
// ===== library: MasterCopy "FB_REOComm" =====

// folder: 04_Heating

FUNCTION_BLOCK "FB_REOComm"   // FB53, SCL
{ S7_Optimized_Access := 'TRUE' }
VERSION : 0.1
   VAR_INPUT
      i_wParameterAdr : Word;   // Address of the parameter to read or write in HEX
      i_wNewValue : Word;   // Value to write to the parameter
      i_wSendStrom : Word;   // Current setpoint (to be sent to REO) 16-Bit 100 % = FFFF H
      i_wSendSpannung : Word;   // Voltage setpoint (to be sent to REO) 16-Bit 100 % = FFFF H
      i_wSendLeistung : Word;   // Power setpoint (to be sent to REO) 16-Bit 100 % = FFFF H
      i_xCurrentPowerMode : Bool;   // 0 = current mode, 1 = power mode
      i_xSendParameter : Bool;   // Trigger to start send parameter sequence
      i_xReadParameter : Bool;   // Trigger to start read parameter sequence
      i_xFreigabeHeiz : Bool;   // Heating enable signal
      i_xResetREO : Bool;   // Trigger to reset REO via parameter mode
      i_xConfigMDW700 : Bool;   // Configuration bit to use the the rigth status byte structure
      i_xConfigWRB : Bool;   // Configuration bit to use the the rigth status byte structure
   END_VAR
   VAR_OUTPUT
      o_REOStatus : "typeREOStatus";   // Structure with REO state and error info
      o_awHWRead : Array[1..4] of Word;   // Read buffer from REO (from DPRD_DAT) [4 WORDs]
      o_wStatusSend : Word;   // Status from the DPWR_DAT call (communication status)
      o_wStatusRead : Word;   // Status from the DPRD_DAT call (communication status)
      o_wReadStrom : Word;   // Measured current from REO (Word 3) Istwert Strom 16 Bit 100% = 8000 H
      o_wReadSpannung : Word;   // Measured voltage from REO (Word 2) Istwert Spannung 16 Bit 100% = 8000 H
      o_wReadLeistung : Word;   // Measured power from REO (Word 2) Istwert Leistung 16 Bit 100% = 4000H
      o_wReadedParameter : Word;   // The parameter value read from REO
      o_xNormalbetrieb : Bool;   // Output for normal operation status
      o_xParameterbetrieb : Bool;   // Output for parameter operation status
      o_xBusy : Bool;   // TRUE when operation in progress
      o_xReadDone : Bool;   // TRUE when Read parameter sequence is done
      o_xResetDone : Bool;   // TRUE when Reset completed successfully
      o_xSendDone : Bool;   // TRUE when Send parameter sequence is done
      o_xError : Bool;   // TRUE if timeout or failure occurred
   END_VAR
   VAR
      TON_TimeResponseOut : TON_TIME;   // Timeout watchdog (e.g., to prevent stuck communication)
      stat_awHWSend : Array[1..4] of Word;   // Internal buffer for writing to REO [4 WORDs]
      iStateWriteParameter : Int;   // Internal state for the write paramter state machine
      iStateReadParameter : Int;   // Internal state for the read paramter state machine
      iStateResetREO : Int;   // Internal state for the reset state machine
      xNormalbetrieb : Bool := TRUE;   // Normal operation mode (standard REO heating control)
      xParameterbetrieb : Bool;   // Parameter operation mode (for parameter read/write/reset)
   END_VAR
   VAR_TEMP
      temp_bySteuerWortError : Byte;
   END_VAR
   VAR CONSTANT
      cCODE : Word := 16#C0DE;   // Constant C0DEH, used in REO protocol as signature
   END_VAR
BEGIN
   (********************************************************************************************************
   Author:     IK
   Date:       2025-04
   Version:    1.1
   *********************************************************************************************************
   Purpose:
   Implements normal mode and parameter mode communication with REO devices via Profinet
   It uses Siemens functions DPRD_DAT and DPWR_DAT to read and write registers from REO
   It also writes status / diagnostic information from REO
   When sending, it sends a sequence of commands: Write Enable, Parameter Write, Release Write Enable,
   Read value and waits for confirmation from the device.
   Use REO Profinet description information documentation to get parameter addresses in Hex

   *********************************************************************************************************
   Modification notes:
   Date:              Name:            Description
   2025-05-19         IK               Added 2 vars: i_xConfigMDW700, i_xConfigWRB
                                       Updated "REO status byte read" block
   *)
   // === Switch to parameter mode when trigger is active ===
   IF (#i_xResetREO
     OR #i_xReadParameter
     OR #i_xSendParameter)
     AND #xNormalbetrieb
   THEN
     // Switch from normal to parameter mode
     #xNormalbetrieb := FALSE;
     #xParameterbetrieb := TRUE;
     #o_xReadDone := FALSE;
     #o_xSendDone := FALSE;
     #o_xResetDone := FALSE;
     #o_xError := FALSE;
   END_IF;

   // === Timeout monitoring for REO system response (5 seconds) ===
   #TON_TimeResponseOut(IN := #xParameterbetrieb
                        AND (#iStateReadParameter <> 0
                        OR #iStateWriteParameter <> 0
                        OR #iStateResetREO <> 0),
                        PT := T#5s);

   IF #TON_TimeResponseOut.Q THEN
     // Timeout: cancel communication and return to normal mode
     #iStateReadParameter := 0;
     #xParameterbetrieb := FALSE;
     #xNormalbetrieb := TRUE;
     #o_xBusy := FALSE;
     #o_xReadDone := FALSE;
     #o_xSendDone := FALSE;
     #o_xError := TRUE;
   END_IF;

   IF #xNormalbetrieb THEN
     //Read from REO
     #o_wStatusRead := INT_TO_WORD(DPRD_DAT(LADDR := "REO_Thyristorsteller_(Phasenanschnitt)~IN_OUT:____8_bytes_1", RECORD => #o_awHWRead));

     IF #i_xCurrentPowerMode THEN
       // Read power and current
       #o_wReadLeistung := #o_awHWRead[2]; // actual power: 4000 = 16384 = 100% max REO power
       #o_wReadStrom := #o_awHWRead[3];    // actual current: 8000 = 32768 = 100% max REO current
     ELSE
       // Read voltage and current
       #o_wReadSpannung := #o_awHWRead[2]; // actual voltage: 8000 = 32768 = 100% max REO voltage
       #o_wReadStrom := #o_awHWRead[3];    // actual current: 8000 = 32768 = 100% max REO current
     END_IF;


     // REO status byte read - read and interpret status byte
     // (various REO operating or fault states depending on error code)
     #temp_bySteuerWortError := #o_awHWRead[4].%B1;
     IF #i_xConfigMDW700 THEN
       CASE #temp_bySteuerWortError OF
         16#00:  // Device not responding
           #o_REOStatus.xReagiertNicht := TRUE;
           #o_REOStatus.xBetriebsbereit := FALSE;
           #o_REOStatus.xParametermodus := FALSE;
           #o_REOStatus.xÜbertemperatur := FALSE;
           #o_REOStatus.xÜberstrom := FALSE;
           #o_REOStatus.xÜberspannung := FALSE;
           #o_REOStatus.xSpitzenStrom := FALSE;
           #o_REOStatus.xUnknowCode := FALSE;
           #o_REOStatus.byREOFehlerCode := #temp_bySteuerWortError;
         16#A5:  // Device ready for operation
           #o_REOStatus.xReagiertNicht := FALSE;
           #o_REOStatus.xBetriebsbereit := TRUE;
           #o_REOStatus.xParametermodus := FALSE;
           #o_REOStatus.xÜbertemperatur := FALSE;
           #o_REOStatus.xÜberstrom := FALSE;
           #o_REOStatus.xÜberspannung := FALSE;
           #o_REOStatus.xSpitzenStrom := FALSE;
           #o_REOStatus.xUnknowCode := FALSE;
           #o_REOStatus.byREOFehlerCode := #temp_bySteuerWortError;
         16#C0:  // Feedback: parameter mode
           #o_REOStatus.xReagiertNicht := FALSE;
           #o_REOStatus.xBetriebsbereit := FALSE;
           #o_REOStatus.xParametermodus := TRUE;
           #o_REOStatus.xÜbertemperatur := FALSE;
           #o_REOStatus.xÜberstrom := FALSE;
           #o_REOStatus.xÜberspannung := FALSE;
           #o_REOStatus.xSpitzenStrom := FALSE;
           #o_REOStatus.xUnknowCode := FALSE;
           #o_REOStatus.byREOFehlerCode := #temp_bySteuerWortError;
         16#70:  // ERROR HOT, overtemperature
           #o_REOStatus.xReagiertNicht := FALSE;
           #o_REOStatus.xBetriebsbereit := FALSE;
           #o_REOStatus.xParametermodus := FALSE;
           #o_REOStatus.xÜbertemperatur := TRUE;
           #o_REOStatus.xÜberstrom := FALSE;
           #o_REOStatus.xÜberspannung := FALSE;
           #o_REOStatus.xSpitzenStrom := FALSE;
           #o_REOStatus.xUnknowCode := FALSE;
           #o_REOStatus.byREOFehlerCode := #temp_bySteuerWortError;
         16#58:  // ERROR OL, overcurrent
           #o_REOStatus.xReagiertNicht := FALSE;
           #o_REOStatus.xBetriebsbereit := FALSE;
           #o_REOStatus.xParametermodus := FALSE;
           #o_REOStatus.xÜbertemperatur := FALSE;
           #o_REOStatus.xÜberstrom := TRUE;
           #o_REOStatus.xÜberspannung := FALSE;
           #o_REOStatus.xSpitzenStrom := FALSE;
           #o_REOStatus.xUnknowCode := FALSE;
           #o_REOStatus.byREOFehlerCode := #temp_bySteuerWortError;
         16#05:  // ERROR UL, overvoltage
           #o_REOStatus.xReagiertNicht := FALSE;
           #o_REOStatus.xBetriebsbereit := FALSE;
           #o_REOStatus.xParametermodus := FALSE;
           #o_REOStatus.xÜbertemperatur := FALSE;
           #o_REOStatus.xÜberstrom := FALSE;
           #o_REOStatus.xÜberspannung := TRUE;
           #o_REOStatus.xSpitzenStrom := FALSE;
           #o_REOStatus.xUnknowCode := FALSE;
           #o_REOStatus.byREOFehlerCode := #temp_bySteuerWortError;
         ELSE  // Unknown status code
           #o_REOStatus.xReagiertNicht := FALSE;
           #o_REOStatus.xBetriebsbereit := FALSE;
           #o_REOStatus.xParametermodus := FALSE;
           #o_REOStatus.xÜbertemperatur := FALSE;
           #o_REOStatus.xÜberstrom := FALSE;
           #o_REOStatus.xÜberspannung := FALSE;
           #o_REOStatus.xSpitzenStrom := FALSE;
           #o_REOStatus.xUnknowCode := TRUE;
           #o_REOStatus.byREOFehlerCode := #temp_bySteuerWortError;
       END_CASE;
     ELSIF #i_xConfigWRB THEN
       CASE #temp_bySteuerWortError OF
         16#00:  // Device not responding
           #o_REOStatus.xReagiertNicht := TRUE;
           #o_REOStatus.xBetriebsbereit := FALSE;
           #o_REOStatus.xParametermodus := FALSE;
           #o_REOStatus.xÜbertemperatur := FALSE;
           #o_REOStatus.xÜberstrom := FALSE;
           #o_REOStatus.xÜberspannung := FALSE;
           #o_REOStatus.xSpitzenStrom := FALSE;
           #o_REOStatus.xUnknowCode := FALSE;
           #o_REOStatus.byREOFehlerCode := #temp_bySteuerWortError;
         16#A5:  // Device ready for operation
           #o_REOStatus.xReagiertNicht := FALSE;
           #o_REOStatus.xBetriebsbereit := TRUE;
           #o_REOStatus.xParametermodus := FALSE;
           #o_REOStatus.xÜbertemperatur := FALSE;
           #o_REOStatus.xÜberstrom := FALSE;
           #o_REOStatus.xÜberspannung := FALSE;
           #o_REOStatus.xSpitzenStrom := FALSE;
           #o_REOStatus.xUnknowCode := FALSE;
           #o_REOStatus.byREOFehlerCode := #temp_bySteuerWortError;
         16#C0:  // Feedback: parameter mode
           #o_REOStatus.xReagiertNicht := FALSE;
           #o_REOStatus.xBetriebsbereit := FALSE;
           #o_REOStatus.xParametermodus := TRUE;
           #o_REOStatus.xÜbertemperatur := FALSE;
           #o_REOStatus.xÜberstrom := FALSE;
           #o_REOStatus.xÜberspannung := FALSE;
           #o_REOStatus.xSpitzenStrom := FALSE;
           #o_REOStatus.xUnknowCode := FALSE;
           #o_REOStatus.byREOFehlerCode := #temp_bySteuerWortError;
         16#70:  // ERROR HOT, overtemperature
           #o_REOStatus.xReagiertNicht := FALSE;
           #o_REOStatus.xBetriebsbereit := FALSE;
           #o_REOStatus.xParametermodus := FALSE;
           #o_REOStatus.xÜbertemperatur := TRUE;
           #o_REOStatus.xÜberstrom := FALSE;
           #o_REOStatus.xÜberspannung := FALSE;
           #o_REOStatus.xSpitzenStrom := FALSE;
           #o_REOStatus.xUnknowCode := FALSE;
           #o_REOStatus.byREOFehlerCode := #temp_bySteuerWortError;
         16#58:  // ERROR OL, overcurrent
           #o_REOStatus.xReagiertNicht := FALSE;
           #o_REOStatus.xBetriebsbereit := FALSE;
           #o_REOStatus.xParametermodus := FALSE;
           #o_REOStatus.xÜbertemperatur := FALSE;
           #o_REOStatus.xÜberstrom := TRUE;
           #o_REOStatus.xÜberspannung := FALSE;
           #o_REOStatus.xSpitzenStrom := FALSE;
           #o_REOStatus.xUnknowCode := FALSE;
           #o_REOStatus.byREOFehlerCode := #temp_bySteuerWortError;
         16#37:  // ERROR UL, overvoltage
           #o_REOStatus.xReagiertNicht := FALSE;
           #o_REOStatus.xBetriebsbereit := FALSE;
           #o_REOStatus.xParametermodus := FALSE;
           #o_REOStatus.xÜbertemperatur := FALSE;
           #o_REOStatus.xÜberstrom := FALSE;
           #o_REOStatus.xÜberspannung := TRUE;
           #o_REOStatus.xSpitzenStrom := FALSE;
           #o_REOStatus.xUnknowCode := FALSE;
           #o_REOStatus.byREOFehlerCode := #temp_bySteuerWortError;
         16#57:  // ERROR PEAK, peak current
           #o_REOStatus.xReagiertNicht := FALSE;
           #o_REOStatus.xBetriebsbereit := FALSE;
           #o_REOStatus.xParametermodus := FALSE;
           #o_REOStatus.xÜbertemperatur := FALSE;
           #o_REOStatus.xÜberstrom := FALSE;
           #o_REOStatus.xÜberspannung := TRUE;
           #o_REOStatus.xSpitzenStrom := TRUE;
           #o_REOStatus.xUnknowCode := FALSE;
           #o_REOStatus.byREOFehlerCode := #temp_bySteuerWortError;
         ELSE  // Unknown status code
           #o_REOStatus.xReagiertNicht := FALSE;
           #o_REOStatus.xBetriebsbereit := FALSE;
           #o_REOStatus.xParametermodus := FALSE;
           #o_REOStatus.xÜbertemperatur := FALSE;
           #o_REOStatus.xÜberstrom := FALSE;
           #o_REOStatus.xÜberspannung := FALSE;
           #o_REOStatus.xSpitzenStrom := FALSE;
           #o_REOStatus.xUnknowCode := TRUE;
           #o_REOStatus.byREOFehlerCode := #temp_bySteuerWortError;
       END_CASE;
     ELSE
       ;   // Optional default: do nothing
     END_IF;

     IF #i_xCurrentPowerMode THEN // Set setpoints and send to REO
       // Power / current mode
       IF #i_xFreigabeHeiz THEN
         // Send voltage and current setpoint, activate Bit 2 (enable)
         #stat_awHWSend[1] := 16#0000;           // must be 0000
         #stat_awHWSend[2] := #i_wSendLeistung;  // setpoint power: 16#FFFF = 65535 = 100% max REO power
         #stat_awHWSend[3] := #i_wSendStrom;     // setpoint current: 16#FFFF = 65535 = 100% REO current
         #stat_awHWSend[4] := 16#4004;           // enable on Bit 2
       ELSE
         // Set everything to 0, disable heating
         #stat_awHWSend[1] := 16#0000;
         #stat_awHWSend[2] := 16#0000;
         #stat_awHWSend[3] := 16#0000;
         #stat_awHWSend[4] := 16#0000;
       END_IF;
     ELSE
       // Voltage / current mode
       IF #i_xFreigabeHeiz THEN
         // Send voltage and current setpoint, activate Bit 2 (enable)
         #stat_awHWSend[1] := 16#0000;           // must be 0000
         #stat_awHWSend[2] := #i_wSendSpannung;  // setpoint voltage: 16#FFFF = 65535 = 100% REO voltage
         #stat_awHWSend[3] := #i_wSendStrom;     // setpoint current: 16#FFFF = 65535 = 100% REO current
         #stat_awHWSend[4] := 16#4004;           // enable on Bit 2
       ELSE
         // Set everything to 0, disable heating
         #stat_awHWSend[1] := 16#0000;
         #stat_awHWSend[2] := 16#0000;
         #stat_awHWSend[3] := 16#0000;
         #stat_awHWSend[4] := 16#0000;           // disable
       END_IF;
     END_IF;


     // Send to REO over DPWR_DAT
     #o_wStatusSend := INT_TO_WORD(DPWR_DAT(LADDR := "REO_Thyristorsteller_(Phasenanschnitt)~IN_OUT:____8_bytes_1", RECORD := #stat_awHWSend));

   ELSIF #xParameterbetrieb THEN
     #o_wStatusRead := INT_TO_WORD(DPRD_DAT(LADDR := "REO_Thyristorsteller_(Phasenanschnitt)~IN_OUT:____8_bytes_1", RECORD => #o_awHWRead));
     CASE #iStateResetREO OF
       0: //Idle: wait for trigger
         IF #i_xResetREO THEN
           // Enable write permission
           #stat_awHWSend[1] := 16#0000;
           #stat_awHWSend[2] := #cCODE;    // Address write key = C0DEH
           #stat_awHWSend[3] := 16#B5C9;   // Write-key for enable = B5E7H
           #stat_awHWSend[4] := 16#8000;   // Mode bits: set mode bit = 1
           #o_wStatusSend := INT_TO_WORD(DPWR_DAT(LADDR := "REO_Thyristorsteller_(Phasenanschnitt)~IN_OUT:____8_bytes_1", RECORD := #stat_awHWSend));
           #iStateResetREO := 1;
           #o_xBusy := TRUE;
         END_IF;

       1: // Wait for confirmation and write reset parameter
         IF #o_awHWRead[1] = 16#0000
           AND #o_awHWRead[2] = #cCODE
           AND #o_awHWRead[3] = 16#B5C9
           AND #o_awHWRead[4] = #cCODE
         THEN
           #stat_awHWSend[1] := 16#0000;
           #stat_awHWSend[2] := 16#9400;   // Address write key = C0DEH
           #stat_awHWSend[3] := 16#C009;   // Write-key for enable = B5E7H
           #stat_awHWSend[4] := 16#8000;   // Mode bits: set mode bit = 1
           #o_wStatusSend := INT_TO_WORD(DPWR_DAT(LADDR := "REO_Thyristorsteller_(Phasenanschnitt)~IN_OUT:____8_bytes_1", RECORD := #stat_awHWSend));
           #iStateResetREO := 2;
         END_IF;

       2: // Wait for confirmation and stop parameter mode
         IF #o_awHWRead[1] = 16#0000
           AND #o_awHWRead[2] = 16#0000
           AND #o_awHWRead[3] = 16#0000
           AND #o_awHWRead[4] = #cCODE
         THEN
           #iStateResetREO := 0;
           #xParameterbetrieb := FALSE;
           #xNormalbetrieb := TRUE;
           #o_xBusy := FALSE;
           #o_xResetDone := TRUE;
         END_IF;
     END_CASE;

     // State machine: read parameter only
     CASE #iStateReadParameter OF
       0: // Idle: wait for trigger and read the parameter
         IF #i_xReadParameter THEN
           #stat_awHWSend[1] := 16#0000;
           #stat_awHWSend[2] := #i_wParameterAdr;
           #stat_awHWSend[3] := 16#0000;
           #stat_awHWSend[4] := 16#8000;
           #o_wStatusSend := INT_TO_WORD(DPWR_DAT(LADDR := "REO_Thyristorsteller_(Phasenanschnitt)~IN_OUT:____8_bytes_1", RECORD := #stat_awHWSend));
           #iStateReadParameter := 1;
           #o_xBusy := TRUE;
         END_IF;

       1: //Wait for response and get the parameter
         IF #o_awHWRead[1] = 16#0000
           AND #o_awHWRead[2] = #i_wParameterAdr
           AND #o_awHWRead[4] = #cCODE
         THEN
           #o_wReadedParameter := #o_awHWRead[3];
           #iStateReadParameter := 0;
           #xParameterbetrieb := FALSE;
           #xNormalbetrieb := TRUE;
           #o_xBusy := FALSE;
           #o_xReadDone := TRUE;
         END_IF;
     END_CASE;

     // State machine: write parameter
     CASE #iStateWriteParameter OF
       0:  // Idle: wait for trigger
         IF #i_xSendParameter THEN
           // Step 1: Send Schreibfreigabe (Write Enable)
           #stat_awHWSend[1] := 16#0000;
           #stat_awHWSend[2] := #cCODE;   // Adresse Schreibschlüssel = C0DEH
           #stat_awHWSend[3] := 16#B5E7;   // Write-key for enable = B5E7H
           #stat_awHWSend[4] := 16#8000;   // Mode bits: set mode bit = 1
           #o_wStatusSend := INT_TO_WORD(DPWR_DAT(LADDR := "REO_Thyristorsteller_(Phasenanschnitt)~IN_OUT:____8_bytes_1", RECORD := #stat_awHWSend));
           #iStateWriteParameter := 1;
           #o_xBusy := TRUE;
         END_IF;

       1:  // Waiting for confirmation of Schreibfreigabe and then send parameter
         IF #o_awHWRead[1] = 16#0000
           AND #o_awHWRead[2] = #cCODE
           AND #o_awHWRead[3] = 16#B5E7
           AND #o_awHWRead[4] = #cCODE
         THEN
           #stat_awHWSend[1] := 16#0000;
           #stat_awHWSend[2] := #i_wParameterAdr OR 16#8000; // Word 2: parameter address with R/W bit; set R/W = 1 (write), for example:
           #stat_awHWSend[3] := #i_wNewValue;  // The new parameter value
           #stat_awHWSend[4] := 16#8000;      // Mode bits (with mode bit = 1)
           #o_wStatusSend := INT_TO_WORD(DPWR_DAT(LADDR := "REO_Thyristorsteller_(Phasenanschnitt)~IN_OUT:____8_bytes_1", RECORD := #stat_awHWSend));
           #iStateWriteParameter := 2;
         END_IF;

       2:  // Waiting for confirmation of send parameter and release write Enable off (Schreibfreigabe aufheben)
         IF #o_awHWRead[1] = 16#0000
           AND #o_awHWRead[2] = (#i_wParameterAdr OR 16#8000)
           AND #o_awHWRead[3] = #i_wNewValue
           AND #o_awHWRead[4] = #cCODE
         THEN
           #stat_awHWSend[1] := 16#0000;
           #stat_awHWSend[2] := 16#C0DE;   // Address write key for release
           #stat_awHWSend[3] := 16#0000;   // Write-key value cleared (0)
           #stat_awHWSend[4] := 16#8000;   // Mode bits remain (with mode bit = 1)
           #o_wStatusSend := INT_TO_WORD(DPWR_DAT(LADDR := "REO_Thyristorsteller_(Phasenanschnitt)~IN_OUT:____8_bytes_1", RECORD := #stat_awHWSend));
           #iStateWriteParameter := 3;
         END_IF;

       3:  // Wait for confirmation and read value
         IF #o_awHWRead[1] = 16#0000
           AND #o_awHWRead[2] = #cCODE
           AND #o_awHWRead[3] = 16#0000
           AND #o_awHWRead[4] = #cCODE
         THEN
           #stat_awHWSend[1] := 16#0000;
           #stat_awHWSend[2] := #i_wParameterAdr;
           #stat_awHWSend[3] := 16#0000;
           #stat_awHWSend[4] := 16#8000;
           #o_wStatusSend := INT_TO_WORD(DPWR_DAT(LADDR := "REO_Thyristorsteller_(Phasenanschnitt)~IN_OUT:____8_bytes_1", RECORD := #stat_awHWSend));
           #iStateWriteParameter := 4;
           #o_xSendDone := TRUE;
         END_IF;

       4:  // Final state: communication sequence finished, reset to idle
         IF #o_awHWRead[1] = 16#0000
           AND #o_awHWRead[2] = #i_wParameterAdr
           AND #o_awHWRead[4] = #cCODE
         THEN
           #o_wReadedParameter := #o_awHWRead[3];

           #iStateWriteParameter := 0;
           #xParameterbetrieb := FALSE;
           #xNormalbetrieb := TRUE;
           #o_xBusy := FALSE;
           #o_xReadDone := TRUE;
         END_IF;
       ELSE
         ;  // Optional default: do nothing
     END_CASE;
   ELSE
     // Optinal default: do nothing
     ;
   END_IF;

   // Outputs
   #o_xNormalbetrieb := #xNormalbetrieb;
   #o_xParameterbetrieb := #xParameterbetrieb;
END_FUNCTION_BLOCK